//==================================================================================================
//								RJM Maszyny sp. z o.o.
//									13.05.2022
//	Obsluga przesuwacza na siłowniku 
//	Siłownik zabieraka plus siłownik przesuwający 
//	Cykl przesuwania: wysun zabierak -> przesun -> schowaj zabierak -> powrót  
// 	v1.0	|| TC v 3.1.4024.22		|| - pierwsza wersja
//==================================================================================================
FUNCTION_BLOCK FB_PrzesuwaczNaSilowniku EXTENDS FB_Podzespol
VAR_INPUT
	stParametry								: DUT_PrzesuwaczNaSilowniku_Parametry;
END_VAR
VAR_OUTPUT
END_VAR
VAR
	bCzujnik0Zabieraka						: ITF_Czujnik;
	bCzujnikMaxZabieraka					: ITF_Czujnik;
	fbElektrozaworZabieraka					: ITF_Elektozawor;
	bCzujnik0Przesuwacza					: ITF_Czujnik;
	bCzujnikMaxPrzesuwacza					: ITF_Czujnik;
	fbElektrozaworPrzesuwacza				: ITF_Elektozawor;
	fbZabierak								: FB_Silownik_Kontrola (	fbCzujnikPozycja0 			:= GVL_Wejscia_IO.bCzujnik0PW_Z, 
																		fbCzujnikPozycjaMax 		:= GVL_Wejscia_IO.bCzujnikMaxPW_Z,
																		fbElektrozawor 				:= GVL_Wyjscia_IO.fbElektrozaworPW_Z);
	fbPrzesuwanie							: FB_Silownik_Kontrola (	fbCzujnikPozycja0 			:= GVL_Wejscia_IO.bCzujnik0PW_N, 
																		fbCzujnikPozycjaMax 		:= GVL_Wejscia_IO.bCzujnikMaxPW_N,
																		fbElektrozawor 				:= GVL_Wyjscia_IO.fbElektrozaworPW_N);

	arrElementyWykonawcze 					: ARRAY [1..GVL_LogowanieBledow_Stale.MAX_ILOSC_ELEMENTOW_NA_PODZESPOL] OF ITF_LogowanieBledow_ElementWykonawczy := 
														[fbZabierak.fbLBKomunikacja, 
														fbPrzesuwanie.fbLBKomunikacja];
	fbLBKomunikacja							: FB_PrzesuwaczNaSilowniku_Komunikacja 
														(arrElementyWykonawcze := arrElementyWykonawcze,
														iIloscPodlementow := 2);

	tonChwilaPoDojechaniu					: TON;
END_VAR

METHOD CyklBazowania_Praca : BOOL
VAR_INPUT
END_VAR
IF (NOT bPierwszePrzejscieBazowanie) THEN
	bPierwszePrzejscieBazowanie				:= TRUE;
	bCyklBazowaniaSkonczony					:= FALSE;
	fbZabierak.PrzesunDoPoczatku			:= TRUE;
END_IF

IF (fbZabierak.NaPoczatku AND NOT fbPrzesuwanie.PrzesuwanieWStronePoczatku) THEN
	fbPrzesuwanie.PrzesunDoPoczatku		:= TRUE;
END_IF

IF (fbPrzesuwanie.NaPoczatku AND fbZabierak.NaPoczatku) THEN
	bPierwszePrzejscieBazowanie				:= FALSE;
	bCyklBazowaniaSkonczony					:= TRUE;
	CyklBazowania_Praca						:= TRUE;
ELSE
	CyklBazowania_Praca						:= FALSE;
END_IF
END_METHOD

METHOD CyklPracy_Praca : BOOL
VAR_INPUT
END_VAR
IF (NOT bPierwszePrzejsciePracy) THEN
	bPierwszePrzejsciePracy					:= TRUE;
	bCyklPracySkonczony						:= FALSE;
	fbZabierak.PrzesunDoKonca				:= TRUE;
	tonChwilaPoDojechaniu.IN				:= FALSE;
	iKrokPracy								:= 1;
END_IF

CASE iKrokPracy OF
	1	:
	IF (fbZabierak.NaKoncu) THEN
		fbPrzesuwanie.PrzesunDoKonca	:= TRUE;
		iKrokPracy							:= 10;
	END_IF
	CyklPracy_Praca							:= TRUE;
	10	:
	IF (fbPrzesuwanie.NaKoncu) THEN
		tonChwilaPoDojechaniu.IN			:= TRUE;
		iKrokPracy							:= 20;
	END_IF
	CyklPracy_Praca							:= TRUE;
	20	:
	IF (tonChwilaPoDojechaniu.Q) THEN
		tonChwilaPoDojechaniu.IN			:= FALSE;
		fbZabierak.PrzesunDoKonca			:= TRUE;
		iKrokPracy							:= 30;
	END_IF
	CyklPracy_Praca							:= TRUE;
	30	:
	IF (fbZabierak.NaPoczatku) THEN
		fbPrzesuwanie.PrzesunDoPoczatku	:= TRUE;
		iKrokPracy							:= 40;
	END_IF
	CyklPracy_Praca							:= TRUE;
	40	:
	IF (fbPrzesuwanie.NaPoczatku) THEN
		iKrokPracy							:= 50;
		bCyklPracySkonczony					:= TRUE;
	END_IF
	CyklPracy_Praca							:= TRUE;
	50	:
		iKrokPracy							:= 0;
		CyklPracy_Praca						:= FALSE;
END_CASE
END_METHOD

METHOD FB_init : BOOL
VAR_INPUT
	bInitRetains : BOOL; // if TRUE, the retain variables are initialized (warm start / cold start)
	bInCopyCode : BOOL;  // if TRUE, the instance afterwards gets moved into the copy code (online change)
	bCzujnik0Zabieraka						: ITF_Czujnik;
	bCzujnikMaxZabieraka					: ITF_Czujnik;
	fbElektrozaworZabieraka					: ITF_Elektozawor;
	bCzujnik0Przesuwacza					: ITF_Czujnik;
	bCzujnikMaxPrzesuwacza					: ITF_Czujnik;
	fbElektrozaworPrzesuwacza				: ITF_Elektozawor;
	
END_VAR

THIS^.bCzujnik0Zabieraka					:= bCzujnik0Zabieraka;			     
THIS^.bCzujnikMaxZabieraka					:= bCzujnikMaxZabieraka;		    
THIS^.fbElektrozaworZabieraka				:= fbElektrozaworZabieraka;		 
THIS^.bCzujnik0Przesuwacza					:= bCzujnik0Przesuwacza;		    
THIS^.bCzujnikMaxPrzesuwacza				:= bCzujnikMaxPrzesuwacza;		  
THIS^.fbElektrozaworPrzesuwacza				:= fbElektrozaworPrzesuwacza;

THIS^.fbZabierak.FB_init (FALSE, FALSE, bCzujnik0Zabieraka, bCzujnikMaxZabieraka, fbElektrozaworZabieraka);
THIS^.fbPrzesuwanie.FB_init (FALSE, FALSE, bCzujnik0Przesuwacza, bCzujnikMaxPrzesuwacza, fbElektrozaworPrzesuwacza);
END_METHOD

METHOD Praca : BOOL
VAR_INPUT
END_VAR
tonChwilaPoDojechaniu (PT := REAL_TO_TIME (stParametry.rCzasNaKoncu));

fbZabierak.Praca ();
fbPrzesuwanie.Praca ();


SUPER^.Praca ();
END_METHOD

METHOD Resetowanie : BOOL
VAR_INPUT
END_VAR
tonChwilaPoDojechaniu.IN					:= FALSE;

SUPER^.Resetowanie ();
END_METHOD

END_FUNCTION_BLOCK

(* stored: Version 1.1.0.1, ProductVersion 3.1.4024.11
   POU FB_PrzesuwaczNaSilowniku: Id {c7ba1278-3548-4e13-8976-321b6c21dbe0}, SpecialFunc None
   Method CyklBazowania_Praca: Id {e436b484-17c0-47ed-a727-72ecc434ecc6}
   Method CyklPracy_Praca: Id {c5710e17-cb66-4931-8ad1-c66f04ccc386}
   Method FB_init: Id {1ce11768-98bf-4742-be1e-5a2040e34f8c}
   Method Praca: Id {50a1e78a-cc3a-4bbd-b431-040552237ed9}
   Method Resetowanie: Id {d30fd266-e071-49ab-aaa8-8763b31c16f0} *)
